(* LS Electric XG5000 project: 6 *)
(* PLC LSPLC *)

(* Comments on direct variables
%MX1	물리필시작
%MX2	물부족알림
%MX3	원두리필시작
%MX4	원두부족알림
%MX5	우유리필시작
%MX6	우유부족알림
*)

PROGRAM NewProgram (* task: 스캔 프로그램 *)
VAR
    on : BOOL;
    t : BOOL;
    timer : TON;
    timer1 : TP;
    timer10 : TON;
    timer11 : TON;
    timer12 : TON;
    timer13 : TON;
    timer14 : TON;
    timer15 : TON;
    timer16 : TON;
    timer2 : TON;
    timer3 : TON;
    timer4 : TON;
    timer5 : TON;
    timer6 : TON;
    timer7 : TON;
    timer8 : TON;
    timer9 : TON;
    가스경고 : BOOL;
    가스센서 : BOOL;
    가스주의 : BOOL;
    경찰신고 : BOOL;
    공기정화 : BOOL;
    매장경고음 : BOOL;
    물 : INT;
    물음표 : BOOL;
    시작 : BOOL;
    알림전송 : BOOL;
    온도 : INT;
    온도경고 : BOOL;
    온도센서 : INT;
    온도위험 : BOOL;
    온도주의 : BOOL;
    우유 : INT;
    원두 : INT;
    유독가스해결 : BOOL;
    유독경고 : BOOL;
    유독안전 : BOOL;
    유독조심 : BOOL;
    유독주의 : BOOL;
    이산화탄소 : INT;
    이상감지 : BOOL;
    일산화탄소 : INT;
    재고물 : INT;
    재고우유 : INT;
    재고원두 : INT;
    전력 : BOOL;
    전력Off : BOOL;
    전력On : BOOL;
    정화완료 : BOOL;
    화재위험 : BOOL;
    화재주의 : BOOL;
    화재진압 : BOOL;
END_VAR
VAR
    _t1 : BOOL;
    _t2 : BOOL;
    _t3 : BOOL;
    _t4 : BOOL;
    _t5 : BOOL;
    _t6 : BOOL;
    _t7 : BOOL;
    _t8 : BOOL;
    _t9 : BOOL;
    _t10 : BOOL;
    _t11 : BOOL;
END_VAR

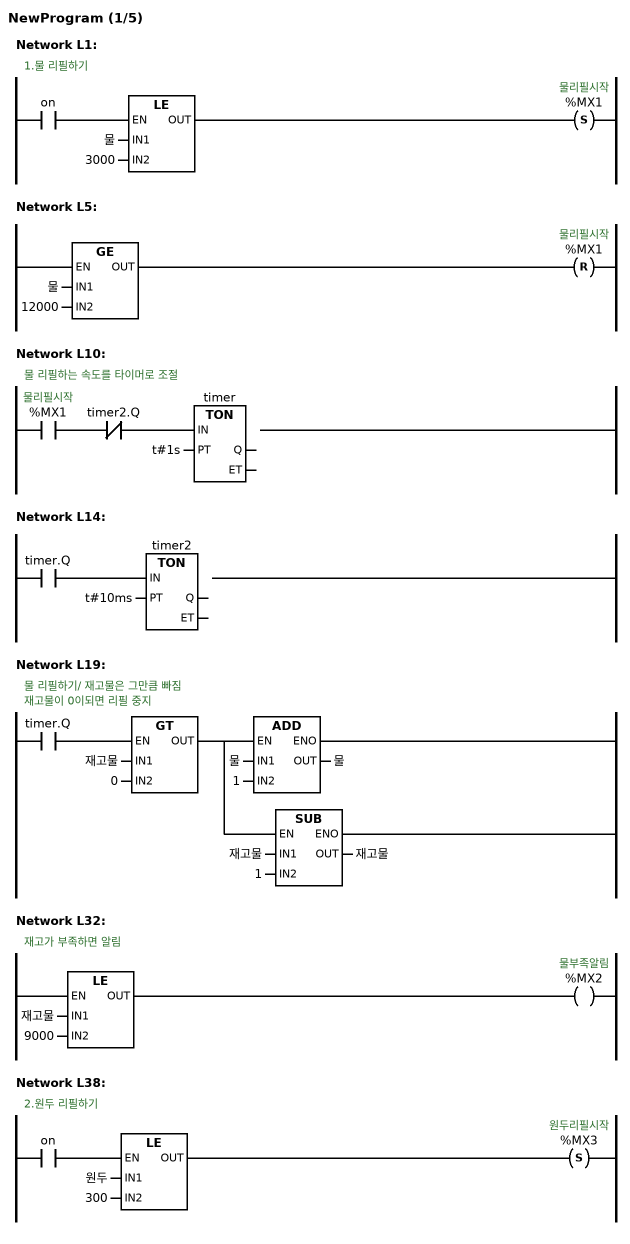
(* 1.물 리필하기 *)
(* Rung L1 *)
IF on THEN _t1 := 물 <= 3000; END_IF;
IF _t1 THEN %MX1 := TRUE; END_IF;
(* Rung L5 *)
IF 물 >= 12000 THEN %MX1 := FALSE; END_IF;
(* 물 리필하는 속도를 타이머로 조절 *)
(* Rung L10 *)
timer(IN := %MX1 AND NOT timer2.Q, PT := t#1s);
(* Rung L14 *)
timer2(IN := timer.Q, PT := t#10ms);
(* 물 리필하기/ 재고물은 그만큼 빠짐 *)
(* 재고물이 0이되면 리필 중지 *)
(* Rung L19 *)
IF timer.Q THEN _t2 := 재고물 > 0; END_IF;
IF _t2 THEN
    물 := 물 + 1;
    재고물 := 재고물 - 1;
END_IF;
(* 재고가 부족하면 알림 *)
(* Rung L32 *)
%MX2 := 재고물 <= 9000;
(* 2.원두 리필하기 *)
(* Rung L38 *)
IF on THEN _t3 := 원두 <= 300; END_IF;
IF _t3 THEN %MX3 := TRUE; END_IF;

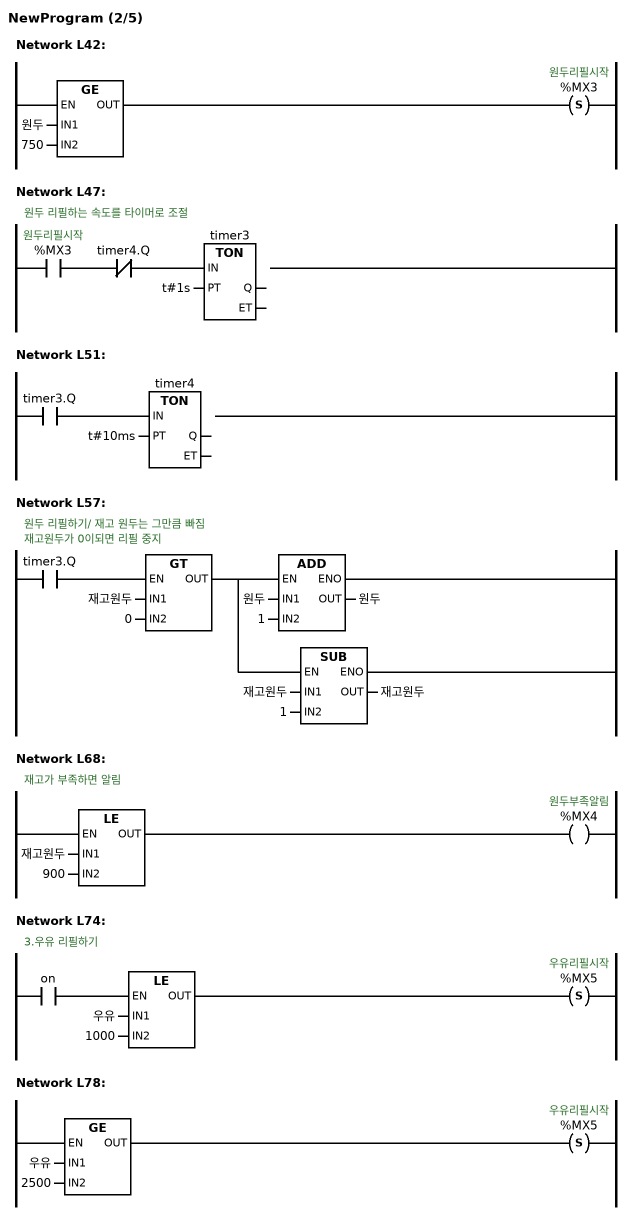
(* Rung L42 *)
IF 원두 >= 750 THEN %MX3 := TRUE; END_IF;
(* 원두 리필하는 속도를 타이머로 조절 *)
(* Rung L47 *)
timer3(IN := %MX3 AND NOT timer4.Q, PT := t#1s);
(* Rung L51 *)
timer4(IN := timer3.Q, PT := t#10ms);
(* 원두 리필하기/ 재고 원두는 그만큼 빠짐 *)
(* 재고원두가 0이되면 리필 중지 *)
(* Rung L57 *)
IF timer3.Q THEN _t4 := 재고원두 > 0; END_IF;
IF _t4 THEN
    원두 := 원두 + 1;
    재고원두 := 재고원두 - 1;
END_IF;
(* 재고가 부족하면 알림 *)
(* Rung L68 *)
%MX4 := 재고원두 <= 900;
(* 3.우유 리필하기 *)
(* Rung L74 *)
IF on THEN _t5 := 우유 <= 1000; END_IF;
IF _t5 THEN %MX5 := TRUE; END_IF;
(* Rung L78 *)
IF 우유 >= 2500 THEN %MX5 := TRUE; END_IF;

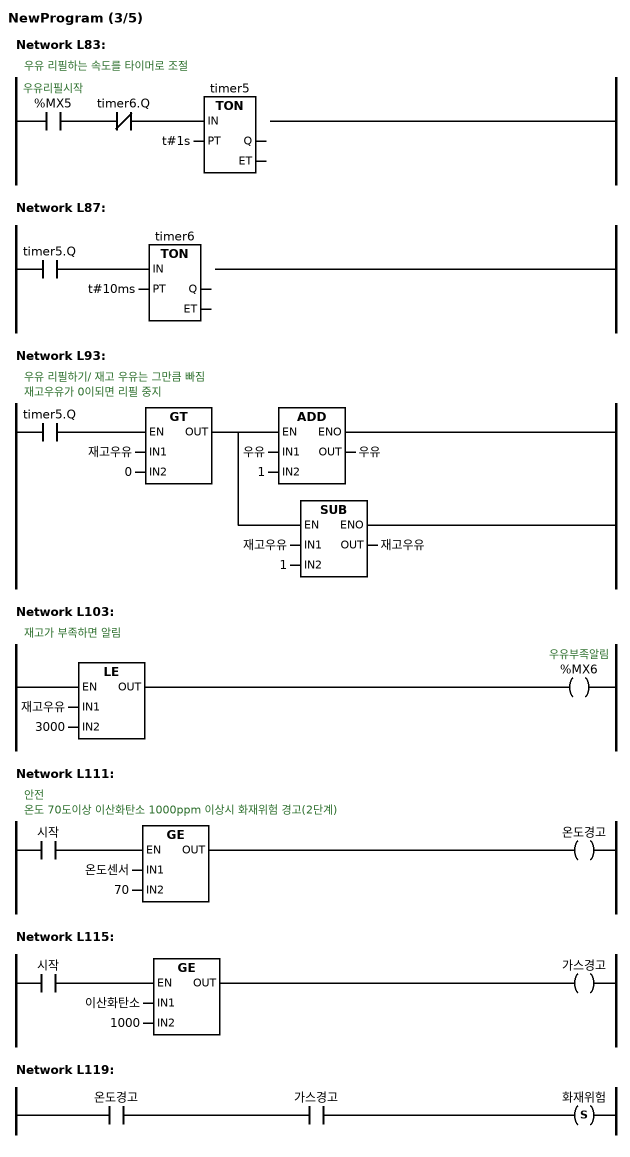
(* 우유 리필하는 속도를 타이머로 조절 *)
(* Rung L83 *)
timer5(IN := %MX5 AND NOT timer6.Q, PT := t#1s);
(* Rung L87 *)
timer6(IN := timer5.Q, PT := t#10ms);
(* 우유 리필하기/ 재고 우유는 그만큼 빠짐 *)
(* 재고우유가 0이되면 리필 중지 *)
(* Rung L93 *)
IF timer5.Q THEN _t6 := 재고우유 > 0; END_IF;
IF _t6 THEN
    우유 := 우유 + 1;
    재고우유 := 재고우유 - 1;
END_IF;
(* 재고가 부족하면 알림 *)
(* Rung L103 *)
%MX6 := 재고우유 <= 3000;
(* 안전 *)
(* 온도 70도이상 이산화탄소 1000ppm 이상시 화재위험 경고(2단계) *)
(* Rung L111 *)
IF 시작 THEN _t7 := 온도센서 >= 70; END_IF;
온도경고 := _t7;
(* Rung L115 *)
IF 시작 THEN _t8 := 이산화탄소 >= 1000; END_IF;
가스경고 := _t8;
(* Rung L119 *)
IF 온도경고 AND 가스경고 THEN 화재위험 := TRUE; END_IF;

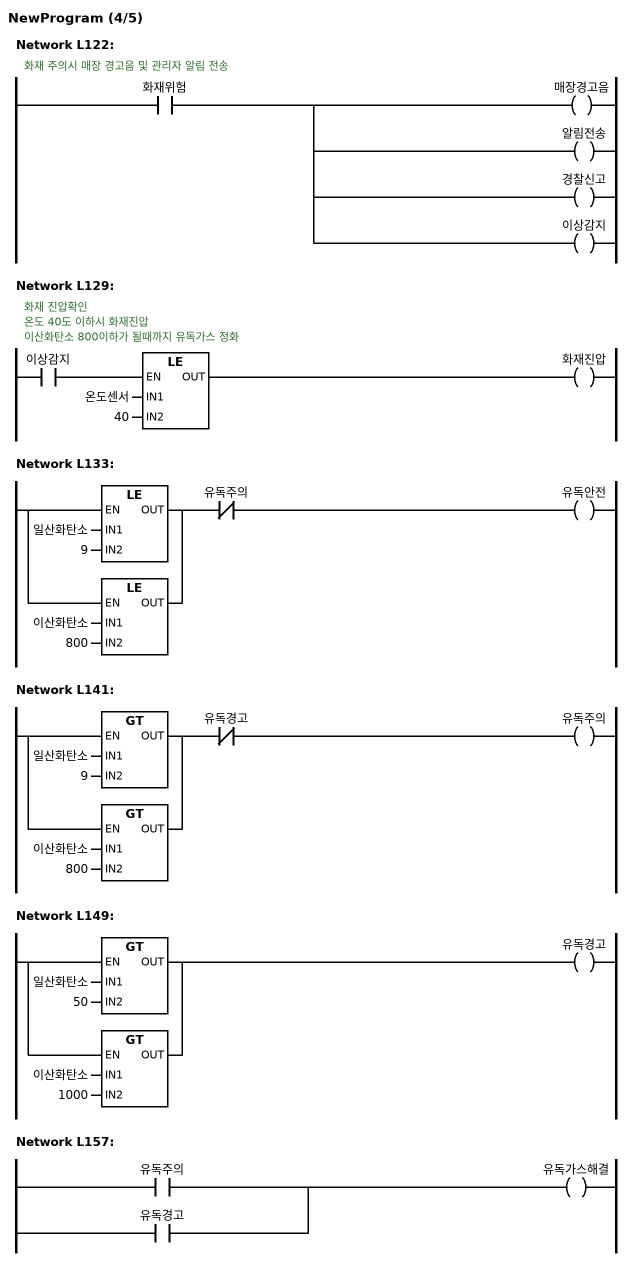
(* 화재 주의시 매장 경고음 및 관리자 알림 전송 *)
(* Rung L122 *)
매장경고음 := 화재위험;
알림전송 := 화재위험;
경찰신고 := 화재위험;
이상감지 := 화재위험;
(* 화재 진압확인 *)
(* 온도 40도 이하시 화재진압 *)
(* 이산화탄소 800이하가 될때까지 유독가스 정화 *)
(* Rung L129 *)
IF 이상감지 THEN _t9 := 온도센서 <= 40; END_IF;
화재진압 := _t9;
(* Rung L133 *)
유독안전 := ((일산화탄소 <= 9) OR (이산화탄소 <= 800)) AND NOT 유독주의;
(* Rung L141 *)
유독주의 := ((일산화탄소 > 9) OR (이산화탄소 > 800)) AND NOT 유독경고;
(* Rung L149 *)
유독경고 := (일산화탄소 > 50) OR (이산화탄소 > 1000);
(* Rung L157 *)
유독가스해결 := 유독주의 OR 유독경고;

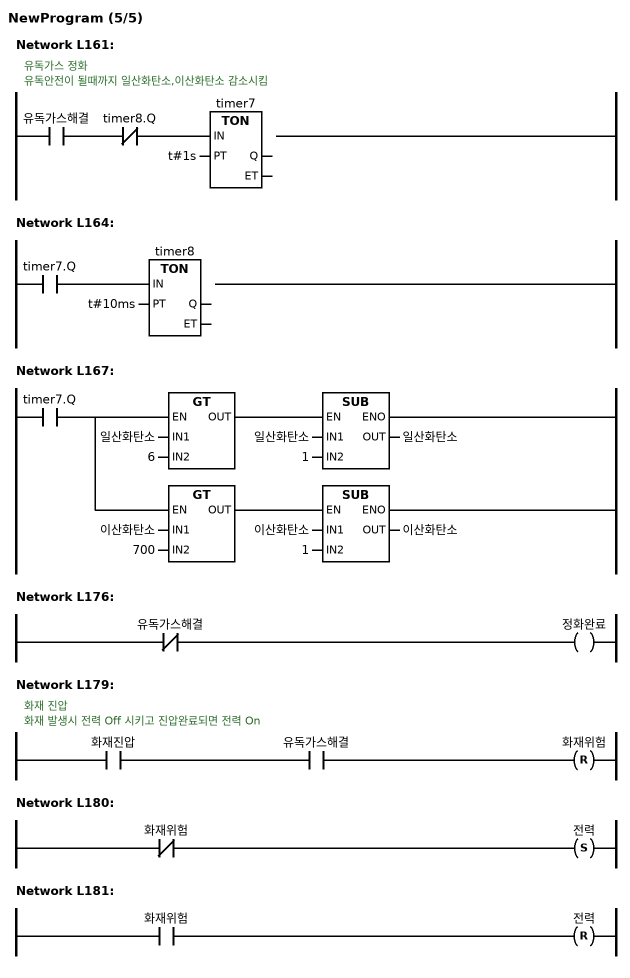
(* 유독가스 정화 *)
(* 유독안전이 될때까지 일산화탄소,이산화탄소 감소시킴 *)
(* Rung L161 *)
timer7(IN := 유독가스해결 AND NOT timer8.Q, PT := t#1s);
(* Rung L164 *)
timer8(IN := timer7.Q, PT := t#10ms);
(* Rung L167 *)
IF timer7.Q THEN _t10 := 일산화탄소 > 6; END_IF;
IF _t10 THEN 일산화탄소 := 일산화탄소 - 1; END_IF;
IF timer7.Q THEN _t11 := 이산화탄소 > 700; END_IF;
IF _t11 THEN 이산화탄소 := 이산화탄소 - 1; END_IF;
(* Rung L176 *)
정화완료 := NOT 유독가스해결;
(* 화재 진압 *)
(* 화재 발생시 전력 Off 시키고 진압완료되면 전력 On *)
(* Rung L179 *)
IF 화재진압 AND 유독가스해결 THEN 화재위험 := FALSE; END_IF;
(* Rung L180 *)
IF NOT 화재위험 THEN 전력 := TRUE; END_IF;
(* Rung L181 *)
IF 화재위험 THEN 전력 := FALSE; END_IF;
END_PROGRAM